{attribute addProperty BoxType "EK1122-0000-0018"}
{attribute addProperty Id "Beckhoff_EJ9xxxsub_EK1100EK1100_179A0949162"}
{attribute addProperty CRC "3683203992"}
{attribute addProperty SizeInBites "16"}
{attribute addProperty SizeInBytes "2"}
TYPE Beckhoff_EJ9xxxEK1122_DB893B98 EXTENDS EK1122_179A0949 :
STRUCT
	{attribute addProperty Name "Beckhoff_EJ9xxxsub_EK1100"}
	Beckhoff_EJ9xxxsub_EK1100 : EK1100_179A0949;
END_STRUCT
END_TYPE

(* stored: Version 1.2.0.0, ProductVersion 3.1.4024.9
   DUT Beckhoff_EJ9xxxEK1122_DB893B98: Id {581034e2-aa1d-44ab-a96b-1bc6ebbb1b7c} *)
